TYPE tstCTCEvent :
STRUCT
	Qualifier 	:USINT; 		// 1 byte event qualifier
	Event 		:teCTCEvent; 	// 2 byte event, converted to enum type
END_STRUCT
END_TYPE

(* stored: Version 1.1.0.1, ProductVersion 3.1.4026.17
   DUT tstCTCEvent: Id {b22a39c8-d824-4ef1-87ec-3259f3477b2c} *)
